(*
	FB_DriveControl manages drive operations by integrating absolute position and velocity control.
    It encapsulates the functionalities of FB_MoveAbsolute for absolute movement and FB_MoveVelocity
    for velocity-based control.
*)
FUNCTION_BLOCK FB_DriveControl
VAR
	_fbMoveAbsolute 		: FB_MoveAbsolute();
	_fbMoveVelocity			: FB_MoveVelocity();

	_fPosition 				: REAL;
	_fVelocity 				: REAL;		
	_bIsPositionReached 	: BOOL := TRUE;		
	
	_fPositionLimitMin 		: REAL := -1E+12;
	_fPositionLimitMax 		: REAL := 1E+12;
	_fAccMax				: REAL := 1E+12;	
	_fTolerance				: REAL := 1E-6;	
END_VAR

(*
    Indicates whether the drive is currently in motion.

    The bIsMoving property returns TRUE if the drive is actively moving toward its target.
*)
PROPERTY bIsMoving : BOOL
GET
bIsMoving := NOT F_Compare(_fVelocity, 0, 1E-3);
END_GET
END_PROPERTY

(*
    Indicates whether the drive has reached its target position.

    This property reflects the internal state of the drive control system.
    It returns TRUE if the drive has achieved the desired position within the specified
    tolerance limits; otherwise, it returns FALSE.
*)
PROPERTY bIsPositionReached : BOOL
GET
bIsPositionReached := _bIsPositionReached;
END_GET
END_PROPERTY

(*
    Maximum Acceleration Limit

    The fAccMax property represents the maximum acceleration permitted for drive movements.
*)
PROPERTY fAccMax : REAL
GET
fAccMax := _fAccMax;
END_GET
SET
_fAccMax := fAccMax;
END_SET
END_PROPERTY

(*
    Actual Drive Position
	
	The fPosition property provides the current position for the drive.
*)
PROPERTY fPosition : REAL
GET
fPosition := _fPosition;
END_GET
SET
_fPosition := fPosition;
END_SET
END_PROPERTY

(*
    Maximum Position Limit
	
	The fPositionLimitMax property defines the upper boundary for the drive's position.
*)
PROPERTY fPositionLimitMax : REAL
GET
fPositionLimitMax := _fPositionLimitMax;
END_GET
SET
_fPositionLimitMax := fPositionLimitMax;
END_SET
END_PROPERTY

(*
    Minimum  Position Limit
	
	The fPositionLimitMax property defines the lower boundary for the drive's position.
*)
PROPERTY fPositionLimitMin : REAL
GET
fPositionLimitMin := _fPositionLimitMin;
END_GET
SET
_fPositionLimitMin := fPositionLimitMin;
END_SET
END_PROPERTY

(*
    Position Tolerance
	
	The fTolerance property defines the acceptable error range for the drive's position.
*)
PROPERTY fTolerance : REAL
GET
fTolerance := _fTolerance;
END_GET
SET
_fTolerance := fTolerance;
END_SET
END_PROPERTY

(*
    Actual Drive Velocity
	
	The fVelocity property provides the current velocity for the drive.
*)
PROPERTY fVelocity : REAL
GET
fVelocity := _fVelocity;
END_GET
SET
_fVelocity := fVelocity;
END_SET
END_PROPERTY

(* 
    Moves the drive to an absolute position.
    
    The MoveAbsolute method commands the drive to move to a specified absolute position with a given velocity,
    acceleration, and deceleration.
*)
METHOD MoveAbsolute
VAR_INPUT
	fPosition 			: REAL;
	fVelocity			: REAL;
	fAcceleration		: REAL;
	fDeceleration   	: REAL;
END_VAR
_fbMoveAbsolute.fPosition := _fPosition;
_fbMoveAbsolute.fVelocity := _fVelocity;

_fbMoveAbsolute(
	fTargetPosition := LIMIT(_fPositionLimitMin, fPosition, _fPositionLimitMax),
	fTargetVelocity := fVelocity,
	fAccMax := fAcceleration,
	fDecMax := fDeceleration,
	fTolerance := _fTolerance);					

_fVelocity := _fbMoveAbsolute.fVelocity;
_fPosition := _fbMoveAbsolute.fPosition;

_bIsPositionReached := F_Compare(fPosition, _fPosition, _fTolerance);
END_METHOD

(* 
    Moves the drive using velocity control.
    
    The MoveVelocity method commands the drive to move with a specified velocity and controls the acceleration
    and deceleration parameters. It also enforces position limits to prevent the drive from exceeding its boundaries.
*)
METHOD MoveVelocity
VAR_INPUT
	fVelocity 			: REAL;
	fAcceleration 		: REAL;
	fDeceleration 		: REAL;
END_VAR
_fbMoveVelocity.fVelocity := _fVelocity;
_fbMoveVelocity.fTargetVelocity := fVelocity;
_fbMoveVelocity.fAccMax := fAcceleration;
_fbMoveVelocity.fDecMax := fDeceleration;	
	
IF _fPositionLimitMax <> 0 AND _fPositionLimitMin <> 0 THEN
	IF _fPosition >= _fPositionLimitMax OR _fPosition <= _fPositionLimitMin THEN
		_fbMoveVelocity.fTargetVelocity := 0;
		_fbMoveVelocity.fAccMax := _fAccMax;
		_fbMoveVelocity.fDecMax := _fAccMax;
	END_IF		
END_IF
	
_fbMoveVelocity();
	
_fVelocity := _fbMoveVelocity.fVelocity;	

_fPosition := _fPosition + _fVelocity * GVL_Core.fbSystem.fDeltaTime * GVL_Core.fbSystem.fTimeScaling;
_bIsPositionReached := F_Compare(fPosition, _fPosition, _fTolerance);
END_METHOD

(* 
    Stops the drive movement.
    
    The Stop method decelerates the drive until it comes to a complete halt using the specified deceleration.
*)
METHOD Stop
VAR_INPUT
	fDeceleration 	: REAL; 
END_VAR

VAR
	fSign 			: REAL;
	fAbsVelocity 	: REAL;
END_VAR
fSign := F_Sign(_fVelocity);
fAbsVelocity := ABS(_fVelocity);

IF fAbsVelocity > fTolerance THEN
	fAbsVelocity := fAbsVelocity - ABS(fDeceleration) * GVL_Core.fbSystem.fDeltaTime * GVL_Core.fbSystem.fTimeScaling;
	fAbsVelocity := LIMIT(0, fAbsVelocity, 3.402823E+38);
	_fVelocity := fAbsVelocity * fSign;	
ELSE
	_fVelocity := 0;
END_IF
END_METHOD

END_FUNCTION_BLOCK

(* stored: Version 1.1.0.1, ProductVersion 3.1.4024.12
   POU FB_DriveControl: Id {dc56c267-b627-0528-22c2-e554d07a3d58}, SpecialFunc None
   Property bIsMoving: Id {73e19af7-d622-0b70-2ddc-0e44cd6fc384}
   Get Get: Id {34506e92-9377-0421-1027-96ada56082df}
   Property bIsPositionReached: Id {8f4cebef-1a01-0cb4-2c9b-b39a96d04003}
   Get Get: Id {0c10a029-e5d5-06f2-3cec-034889a553cf}
   Property fAccMax: Id {cbc5a371-916a-036a-36ba-312db2ce89eb}
   Get Get: Id {833d2f7c-2121-0dd5-0aa5-7a1eceeb4fdd}
   Set Set: Id {76e4d8b1-b2da-0ecb-0ba6-0535e0f7b081}
   Property fPosition: Id {059e2d77-deb5-0e01-35eb-131abdf4b729}
   Get Get: Id {c931bd96-dda6-09e5-0854-c99182dbe955}
   Set Set: Id {a61cb87a-1253-04f5-0264-b5565a3ea35a}
   Property fPositionLimitMax: Id {fa7b5bed-e9f1-00b0-2694-7fd5d07b2165}
   Get Get: Id {30579d96-7fa8-044c-298c-52dedd9f6e10}
   Set Set: Id {a9b2a74c-3cbd-09e3-2f97-44ede0ae5a1c}
   Property fPositionLimitMin: Id {4154ad98-973b-0b01-179b-6e880cfaa026}
   Get Get: Id {328a948d-81a9-0388-23f2-1bd27eef4930}
   Set Set: Id {4b6b1684-e68e-0cb9-2478-e4b4232650c2}
   Property fTolerance: Id {77ed7496-39fc-05df-196f-13e6115f8789}
   Get Get: Id {0b58fdbc-bb13-0dbf-21d4-f64d65aea821}
   Set Set: Id {0d15f425-9688-0993-1418-3e88fc0cd39d}
   Property fVelocity: Id {51a8cd0e-a3fd-0189-3eb3-54ee4c21bc32}
   Get Get: Id {7bedfb7c-fa77-0e4d-1c13-7cb05df11252}
   Set Set: Id {2e195c7c-d9e4-08a9-2399-1b5019693925}
   Method MoveAbsolute: Id {be210045-6d8a-0f76-38f1-25a7a667b3e2}
   Method MoveVelocity: Id {67902dcb-c091-0097-0c26-f6a25649f8cd}
   Method Stop: Id {989f0471-080e-05a5-05a7-9d4740e325c8} *)
